{attribute 'GeneratedUsingTerminal: EL3692-0000-0020'}
{attribute addProperty BoxType "EL3692-0000-0020"}
{attribute addProperty Id "ControlAT %Q*Control_E49DBA1B4"}
{attribute addProperty CRC "4124687394"}
{attribute addProperty Size "4"}
TYPE SAI_Range_Control_Channel_F5D9BC22 EXTENDS TcoIo.OutputBase_10CEE7DE : STRUCT
    {attribute addProperty Name "Control"}
    Control AT %Q* : Control_E49DBA1B;
END_STRUCT
END_TYPE

(* stored: Version 1.2.0.0, ProductVersion 3.1.4024.11
   DUT SAI_Range_Control_Channel_F5D9BC22: Id {41244d50-b102-0d19-330e-219bd143940e} *)
